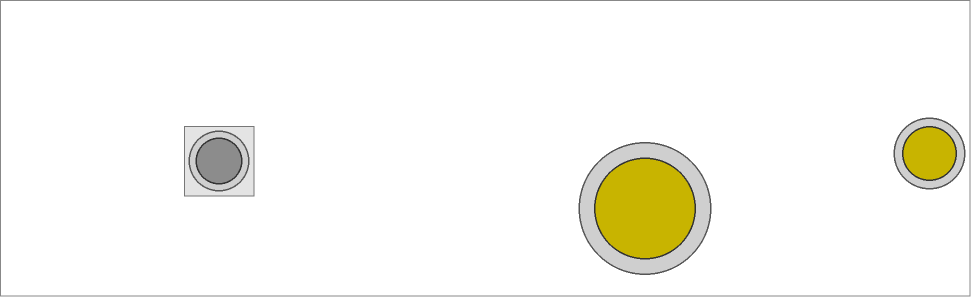
VISUALIZATION Visualization  // 971x297
    PushSwitch (184,126 70x70), variable: MAIN.bHmiButton, behaviour: TOGGLE, style: Switch-PushSwitch-Gray
    Lamp1 (568,120 154x177), variable: MAIN.bMainMotor, style: Lamp-Lamp1-Yellow
    Lamp1 (888,111 83x85), variable: MAIN.bHardwareButton, style: Lamp-Lamp1-Yellow
END_VISUALIZATION

(* stored: Version 1.1.0.1
   Visu Visualization: Id {72c10167-2b27-44e6-ad00-adeb974fe7b1} *)
